(* IEC 61131-3 sources: ATCMcontrol_Engineering/src/COM/softing/fc/AddOns/Softing/4CPCTarget/Libs/ATCM_IEC1131_3/table_30, 12 files *)

(* ---- add_dt_time.st ---- *)
(*[[
    UserURL= "ATCM:ADD_DT_TIME.htm"
]]*)

FUNCTION ADD_DT_TIME : DT
VAR_INPUT
    IN1  : DT;
    IN2  : TIME;
END_VAR
inline +
END_FUNCTION

(* ---- add_time.st ---- *)
(*[[
    UserURL= "ATCM:ADD_TIME.htm"
]]*)

FUNCTION ADD_TIME : TIME
VAR_INPUT
    IN1 : TIME;
    IN2 : TIME;
END_VAR

inline +

END_FUNCTION

(* ---- add_tod_time.st ---- *)
(*[[
    UserURL= "ATCM:ADD_TOD_TIME.htm"
]]*)

FUNCTION ADD_TOD_TIME : TOD
VAR_INPUT
    IN1 : TOD;
    IN2 : TIME;
END_VAR
inline +
END_FUNCTION

(* ---- concat_date_tod.st ---- *)
(*[[
    UserURL= "ATCM:CONCAT_DATE_TOD.htm"
]]*)

FUNCTION CONCAT_DATE_TOD : DT
VAR_INPUT
    IN1 : DATE;
    IN2 : TOD;
END_VAR

inline{Utils.concat_date_tod(%1,%2)}

END_FUNCTION

(* ---- divtime.st ---- *)
(*[[
    UserURL= "ATCM:DIVTIME.htm"
]]*)

FUNCTION DIVTIME : TIME
VAR_INPUT
    IN1 : TIME;
    IN2 : ANY_NUM;
END_VAR

inline /

END_FUNCTION

(* ---- multime.st ---- *)
(*[[
    UserURL= "ATCM:MULTIME.htm"
]]*)

FUNCTION MULTIME : TIME
VAR_INPUT
    IN1 : TIME;
    IN2 : ANY_NUM;
END_VAR

inline *

END_FUNCTION

(* ---- sub_date_date.st ---- *)
(*[[
    UserURL= "ATCM:SUB_DATE_DATE.htm"
]]*)

FUNCTION SUB_DATE_DATE : TIME
VAR_INPUT
    IN1 : DATE;
    IN2 : DATE;
END_VAR

inline -

END_FUNCTION

(* ---- sub_dt_dt.st ---- *)
(*[[
    UserURL= "ATCM:SUB_DT_DT.htm"
]]*)

FUNCTION SUB_DT_DT : TIME
VAR_INPUT
    IN1 : DT;
    IN2 : DT;
END_VAR

inline -

END_FUNCTION

(* ---- sub_dt_time.st ---- *)
(*[[
    UserURL= "ATCM:SUB_DT_TIME.htm"
]]*)

FUNCTION SUB_DT_TIME : DT
VAR_INPUT
    IN1 : DT;
    IN2 : TIME;
END_VAR

inline -

END_FUNCTION

(* ---- sub_time.st ---- *)
(*[[
    UserURL= "ATCM:SUB_TIME.htm"
]]*)

FUNCTION SUB_TIME : TIME
VAR_INPUT
    IN1 : TIME;
    IN2 : TIME;
END_VAR

inline -

END_FUNCTION

(* ---- sub_tod_time.st ---- *)
(*[[
    UserURL= "ATCM:SUB_TOD_TIME.htm"
]]*)

FUNCTION SUB_TOD_TIME : TOD
VAR_INPUT
    IN1 : TOD;
    IN2 : TIME;
END_VAR

inline -

END_FUNCTION

(* ---- sub_tod_tod.st ---- *)
(*[[
    UserURL= "ATCM:SUB_TOD_TOD.htm"
]]*)

FUNCTION SUB_TOD_TOD : TIME
VAR_INPUT
    IN1 : TOD;
    IN2 : TOD;
END_VAR

inline -

END_FUNCTION
